// TwinCAT 3 PLC project Main
// ProgramVersion: 3.1.4024.0
// libraries:
//   Tc2_Standard, * (Beckhoff Automation GmbH)
//   Tc2_System, * (Beckhoff Automation GmbH)
//   Tc2_Utilities, * (Beckhoff Automation GmbH)
//   Tc3_Module, * (Beckhoff Automation GmbH)
//   TcUnit, * (www.tcunit.org)
//   mobject-graph,0.16.0,mobject
// project tree:
//   / PlcTask.TcTTO (not stored)
//   POUs/ MAIN.TcPOU (not stored)
//   Tests/Mocks/ TestNode.TcPOU
//   Tests/ NodePrototype_TestSuite.TcPOU, NodeHost_TestSuite.TcPOU

// ---- Tests/Mocks/TestNode.TcPOU
FUNCTION_BLOCK INTERNAL TestNode EXTENDS Node

METHOD PUBLIC Clone : I_Node
VAR_INPUT
END_VAR
END_METHOD

METHOD PROTECTED OnExecute
END_METHOD

METHOD SetId
VAR_INPUT
    Id : T_MaxString;
END_VAR
SUPER^._id := Id;
END_METHOD

END_FUNCTION_BLOCK

// ---- Tests/NodePrototype_TestSuite.TcPOU
FUNCTION_BLOCK NodePrototype_TestSuite EXTENDS TcUnit.FB_TestSuite
VAR
END_VAR

TestNodeReturnsExpected();
TestPathReturnsExpected();

METHOD TestNodeReturnsExpected
VAR
    node : TestNode;
	prototype : NodePrototype('TestPath', node);
	expected : I_Node;
	actual : I_Node;
END_VAR
TEST('TestNodeReturnsExpected');

expected := node;
actual := prototype.Node;

AssertEquals(
	Expected := expected, 
	Actual := actual,
	Message := 'Did not produce the expected result'
);

TEST_FINISHED();
END_METHOD

METHOD TestPathReturnsExpected
VAR
    node : TestNode;
	prototype : NodePrototype('TestPath', node);
	expected : T_MAXSTRING := 'TestPath';
	actual : T_MAXSTRING;
END_VAR
TEST('TestPathReturnsExpected');

actual := prototype.Path;

AssertEquals_STRING(
	Expected := expected, 
	Actual := actual,
	Message := 'Did not produce the expected result'
);

TEST_FINISHED();
END_METHOD

END_FUNCTION_BLOCK

// ---- Tests/NodeHost_TestSuite.TcPOU
FUNCTION_BLOCK NodeHost_TestSuite EXTENDS TcUnit.FB_TestSuite
VAR
END_VAR

TestHasNodesAfterInit();
TestHasNodesAfterAdding();
TestRemoveNode();
TestTryGetNodeById();

METHOD TestHasNodesAfterAdding
VAR
    node : TestNode;
	host : NodeHost(0, 0);
	actual : BOOL;
END_VAR
TEST('TestHasNodesAfterAdding');

host.AddNode(Node);

actual := host.HasNodes;

AssertTrue(
	Condition := actual, 
	Message := 'Did not produce the expected result'
);

TEST_FINISHED();
END_METHOD

METHOD TestHasNodesAfterInit
VAR
	host : NodeHost(0, 0);
	actual : BOOL;
END_VAR
TEST('TestHasNodesAfterInit');

actual := host.HasNodes;

AssertFalse(
	Condition := actual, 
	Message := 'Did not produce the expected result'
);

TEST_FINISHED();
END_METHOD

METHOD TestRemoveNode
VAR CONSTANT
    NODES_TO_TEST : INT := 10;
END_VAR
VAR
    nodes : ARRAY [1..NODES_TO_TEST] OF TestNode;
    index : INT;
	host : NodeHost(0, 0);
	actual : BOOL;
END_VAR
TEST('TestRemoveNode');

FOR index := 1 TO NODES_TO_TEST BY 1 DO
    nodes[index].SetId(TO_STRING(index));
    host.AddNode(nodes[index]);
END_FOR

FOR index := 1 TO NODES_TO_TEST BY 1 DO
    host.RemoveNode(nodes[index]);
END_FOR

actual := host.HasNodes;

AssertFalse(
	Condition := actual, 
	Message := 'Did not produce the expected result'
);

TEST_FINISHED();
END_METHOD

METHOD TestTryGetNodeById
VAR CONSTANT
    NODES_TO_TEST : INT := 10;
END_VAR
VAR
    nodes : ARRAY [1..NODES_TO_TEST] OF TestNode;
    guids : ARRAY [1..NODES_TO_TEST] OF T_MaxString := ['54E2a4bf-7608-4ba2-b7a0-cc0d122ca5b9',
                                                        '36b64dc1-33b7-4132-ace0-8e026acf58da',
                                                        '9E922f40-7a98-462a-9571-b394f5afad1e',
                                                        '5dee9f3f-35b7-4e74-8e59-b921d102c5b9',
                                                        '55ee8e9d-3a44-4E6b-81aa-9c2f4ce65bce',
                                                        '1192e990-56ea-4185-a4ad-a2e7413437b3',
                                                        'dafdbd2c-5f76-403d-8f89-c6aec472b210',
                                                        '4e1a0640-6b80-4880-91d1-47f8fc8f9be7',
                                                        '5f950222-f5dd-4bce-914e-b4a0d60d2e77',
                                                        '17190E2e-6ca3-40a2-80c5-b209cf3c06a5'];
    index : INT;	
    host : NodeHost(0, 0);
    foundNode : I_Node;
	actual : BOOL;
END_VAR
TEST('TestTryGetNodeById');

FOR index := 1 TO NODES_TO_TEST BY 1 DO
    nodes[index].SetId(guids[index]);
    host.AddNode(nodes[index]);
END_FOR

actual := host.TryGetNodeById('5dee9f3f-35b7-4e74-8e59-b921d102c5b9', foundNode);

AssertTrue(
	Condition := actual, 
	Message := 'Did not produce the expected result'
);

TEST_FINISHED();
END_METHOD

END_FUNCTION_BLOCK
